FUNCTION FC_Check_ACK : BOOL
VAR_INPUT
	I_sString : REFERENCE TO T_MaxString;
END_VAR
VAR
	stringPos	: INT;
END_VAR

stringPos := FIND(I_sString, ACK);
IF stringPos <> 0 THEN
	I_sString := MID(I_sString, LEN(I_sString), stringPos+1);
	FC_Check_ACK := TRUE;
ELSE
	FC_Check_ACK := FALSE;
END_IF

END_FUNCTION

(* stored: Version 1.1.0.1, ProductVersion 3.1.4024.15
   POU FC_Check_ACK: Id {409ebcc3-ff01-45a0-b2e5-de3116ef15d1}, SpecialFunc None *)
